// TIA Portal V17 export
// export: Created 2023-04-04T13:27:25.6384543Z, ExportSetting WithDefaults, DisplayName Totally Integrated Automation Portal, DisplayVersion V17, DisplayName TIA Portal Openness, DisplayVersion V17, DisplayName TIA Portal Version Control Interface, DisplayVersion V17, DisplayName STEP 7 Professional, DisplayVersion V17, DisplayName STEP 7 Safety, DisplayVersion V17, DisplayName WinCC Advanced, DisplayVersion V17
DATA_BLOCK "PRG_HBW_Axis_Horizontal_DB"   // DB18
AUTHOR : A.Schaefer
VERSION : 0.1
// stored: AutoNumber true, DBAccessibleFromOPCUA true, DBAccessibleFromWebserver true, InstanceOfName PRG_HBW_Axis_Horizontal, InstanceOfType FB
"PRG_HBW_Axis_Horizontal"
   // VAR
   //    lx_Init { ExternalAccessible := 'False'; ExternalVisible := 'False'; ExternalWritable := 'False'} : Bool;
   //    lfb_Horizontal_Axis { ExternalAccessible := 'False'; ExternalVisible := 'False'; ExternalWritable := 'False'} : "FB_Axis_Auto";
   // END_VAR
BEGIN
END_DATA_BLOCK
